ABB RobotStudio station: IRB120_GroupL_20170908-110615.rsstn

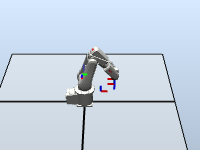
Station Station (saved by RobotStudio 6.5.7502.1049)
Controller MTRN4230
  mechanical unit ROB_1: IRB120_3_58__01, 6 joints, base frame (0, 0, 0) mm
Layout (positions relative to the parent item):
  - IRB120_3_58__01 [mechanism, from Robots\IRB120_3_58_G_01.rslib] at (0, 0, 0) mm; joint values [0.1225, 0.318, 0.5796, 0, 0.6732, 0.1225] (rad or m)
Targets, tools, work objects and paths stored in the station, written as RAPID:
! task RobControl
MODULE MTRN4230_Move_Sample
  PROC MoveJSample()
    MoveJ pConvHome,v100,fine,tSCup;
  ENDPROC
  PROC MoveLSample()
    MoveL Offs(pTableHome, 0, 0, 100),v100,fine,tSCup;
  ENDPROC
  PROC MainMove()
  ENDPROC
ENDMODULE

! task RobControl
MODULE MTRN4230_IO_Sample
  PROC MainIO()
  ENDPROC
  PROC TurnVacOff()
    SetDO DO10_1,0;
  ENDPROC
  PROC TurnConOff()
    SetDO DO10_3,0;
  ENDPROC
  PROC TurnVacOn()
    SetDO DO10_1,1;
  ENDPROC
  PROC TurnConOnSafely()
    SetDO DO10_3,1;
    SetDO DO10_3,0;
  ENDPROC
ENDMODULE

! task RobControl
MODULE MTRN_Rob_Data
  CONST robtarget pConvHome:=[[0,409,22],[0,-0.7071068,0.7071068,0],[0,0,0,0],[9E+09,9E+09,9E+09,9E+09,9E+09,9E+09]];
  PERS tooldata tSCup:=[TRUE,[[0,0,65],[1,0,0,0]],[0.5,[0,0,20],[1,0,0,0],0,0,0]];
  PERS wobjdata wTable:=[FALSE,TRUE,"",[[175,0,147],[1,0,0,0]],[[0,0,0],[1,0,0,0]]];
  PERS wobjdata wConv:=[FALSE,TRUE,"",[[50,184,22],[0.5,-0.5,0.5,0.5]],[[1,1,1],[1,0,0,0]]];
  CONST jointtarget jtCalibPos:=[[-90,0,0,0,0,0],[9E+09,9E+09,9E+09,9E+09,9E+09,9E+09]];
ENDMODULE

! task RobControl
MODULE MTRN_Rob_Proc
  PROC MoveToCalibPos()
    MoveAbsJ jtCalibPos,v400,fine,tool0;
  ENDPROC
ENDMODULE

